TYPE TestResults :
STRUCT
	Passed		: BOOL;
	Message		: STRING(255);
END_STRUCT
END_TYPE

(* stored: Version 1.1.0.1
   DUT TestResults: Id {359f6d4c-c185-4772-9f70-f81130d97630} *)
